FUNCTION_BLOCK ShrunkMatrixAccessor EXTENDS MatrixAccessor
VAR_INPUT
END_VAR
VAR_OUTPUT
END_VAR
VAR
	RowRemoved_ : UINT;
	ColRemoved_ : UINT;
END_VAR

//Total number of columns in this matrix
PROPERTY PUBLIC Cols : UINT
GET
IF NOT __ISVALIDREF(M_) THEN
	Cols := 0;
	LogWarning('%s Attempted Cols access using uninitialized Matrix Accessor');
ELSIF M_.Cols > 0 THEN
	Cols := M_.Cols-1;
ELSE
	Cols := 0;
END_IF
END_GET
END_PROPERTY

METHOD PUBLIC Init
VAR_INPUT
	M : REFERENCE TO Matrix;
	RowRemoved : UINT;
	ColRemoved : UINT;
END_VAR
Init_(M);
RowRemoved_ := RowRemoved;
ColRemoved_ := ColRemoved;
END_METHOD

//Total number of rows in this matrix
PROPERTY PUBLIC Rows : UINT
GET
IF NOT __ISVALIDREF(M_) THEN
	Rows := 0;
	LogWarning('%s Attempted Rows access using uninitialized Matrix Accessor');
ELSIF M_.Rows > 0 THEN
	Rows := M_.Rows-1;
ELSE
	Rows := 0;
END_IF
END_GET
END_PROPERTY

METHOD PROTECTED This2Parent : UINT
VAR_INPUT
	Index : UINT;
END_VAR
VAR
	ThisR : UINT;
	ThisC : UINT;
END_VAR
IF NOT __ISVALIDREF(M_) THEN
	LogWarning('%s Attempted This2Parent calculation using uninitialized Matrix Accessor');
	This2Parent := 0;
	RETURN;
END_IF

IC2RC(Index,Cols,Row => ThisR, Col => ThisC);

This2Parent := RCC2I(ThisR+BOOL_TO_UINT(RowRemoved_<=ThisR),ThisC+BOOL_TO_UINT(ColRemoved_<=ThisC),M_.Cols);
END_METHOD

END_FUNCTION_BLOCK

(* stored: Version 1.1.0.1, ProductVersion 3.1.4024.9
   POU ShrunkMatrixAccessor: Id {f0bfcb10-4309-028c-1405-e53184e0781f}, SpecialFunc None
   Folder Initializers: Id {45740341-dbbb-08f6-3340-7857963b9e64}
   Folder Overrides: Id {967fd700-932b-0466-3705-406f25b48dc3}
   Property Cols: Id {f3e7e618-58e0-0e81-02db-fc0fc539f3ee}
   Get Get: Id {1c7f5a4f-f036-0f00-0aab-5b1385b88ad9}
   Method Init: Id {9d266aca-2413-0651-3a78-fd0697cc15bb}
   Property Rows: Id {7c4ed6f3-3d01-028d-1d23-3c66c33be3ce}
   Get Get: Id {f08fb378-8ee8-0f98-35a7-7b3a88876ac2}
   Method This2Parent: Id {0063716a-7aa7-0c6f-17df-1e2c021e63a3} *)
